// TIA Portal V17 export
// export: Created 2023-04-04T07:47:19.0202883Z, ExportSetting WithDefaults, DisplayName Totally Integrated Automation Portal, DisplayVersion V17 Update 4, DisplayName TIA Portal Openness, DisplayVersion V17 Update 4, DisplayName TIA Portal Version Control Interface, DisplayVersion V17, DisplayName STEP 7 Professional, DisplayVersion V17 Update 4, DisplayName STEP 7 Safety, DisplayVersion V17, DisplayName WinCC Professional, DisplayVersion V17 Update 4
FUNCTION "BMS 1 (F)" : Void   // FC21, LAD
TITLE = ModBus TCP for CATL Battery
{ S7_Optimized_Access := 'TRUE' }
VERSION : 0.1
// stored: AutoNumber false, IsIECCheckEnabled false, SetENOAutomatically false, UDAEnableTagReadback false
   VAR_TEMP
      xSpare : Bool;
      BBwAlm1 : Word;
      BBwWarn1 : Word;
      BR01wAlm1 : Word;
      BR01wAlm2 : Word;
      BR01wAlm3 : Word;
      BR01wWarn1 : Word;
      BR02wAlm1 : Word;
      BR02wAlm2 : Word;
      BR02wAlm3 : Word;
      BR02wWarn1 : Word;
      BR03wAlm1 : Word;
      BR03wAlm2 : Word;
      BR03wAlm3 : Word;
      BR03wWarn1 : Word;
      BR04wAlm1 : Word;
      BR04wAlm2 : Word;
      BR04wAlm3 : Word;
      BR04wWarn1 : Word;
      BR05wAlm1 : Word;
      BR05wAlm2 : Word;
      BR05wAlm3 : Word;
      BR05wWarn1 : Word;
      BR06wAlm1 : Word;
      BR06wAlm2 : Word;
      BR06wAlm3 : Word;
      BR06wWarn1 : Word;
      BR07wAlm1 : Word;
      BR07wAlm2 : Word;
      BR07wAlm3 : Word;
      BR07wWarn1 : Word;
      BR08wAlm1 : Word;
      BR08wAlm2 : Word;
      BR08wAlm3 : Word;
      BR08wWarn1 : Word;
      BR09wAlm1 : Word;
      BR09wAlm2 : Word;
      BR09wAlm3 : Word;
      BR09wWarn1 : Word;
      BR10wAlm1 : Word;
      BR10wAlm2 : Word;
      BR10wAlm3 : Word;
      BR10wWarn1 : Word;
   END_VAR
BEGIN

REGION Network 1: Function Modbus Client
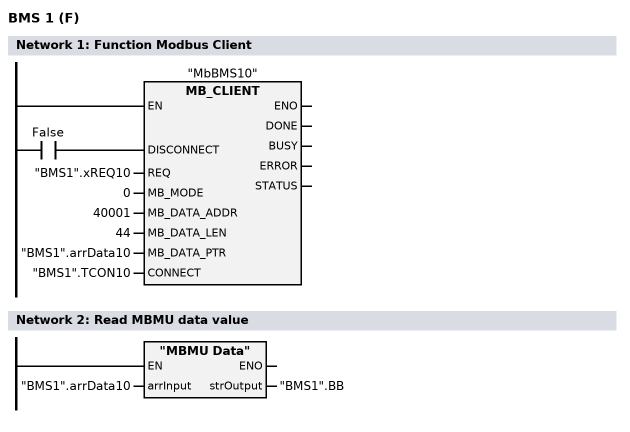
   RUNG wire#powerrail
      "MbBMS10".MB_CLIENT(DISCONNECT := wire#w1, REQ := "BMS1".xREQ10, MB_MODE := 0, MB_DATA_ADDR := 40001, MB_DATA_LEN := 44, MB_DATA_PTR := "BMS1".arrData10, CONNECT := "BMS1".TCON10, DONE =>, BUSY =>, ERROR =>, STATUS =>)
   END_RUNG
   RUNG wire#powerrail
      Contact( False )
   END_RUNG wire#w1
   // the same network as SCL:
   "MbBMS10"(DISCONNECT := False,   // MB_CLIENT
             REQ := "BMS1".xREQ10,
             MB_MODE := 0,
             MB_DATA_ADDR := 40001,
             MB_DATA_LEN := 44,
             MB_DATA_PTR := "BMS1".arrData10,
             CONNECT := "BMS1".TCON10);
END_REGION

REGION Network 2: Read MBMU data value
   RUNG wire#powerrail
      "MBMU Data"(arrInput := "BMS1".arrData10, strOutput => "BMS1".BB)
   END_RUNG
   // the same network as SCL:
   "MBMU Data"(arrInput := "BMS1".arrData10, strOutput => "BMS1".BB);
END_REGION
END_FUNCTION
